PROGRAM Programm
VAR
	Alarm_Off_Time: TIME := T#3S;
	Alarm_0: Alarm;
END_VAR

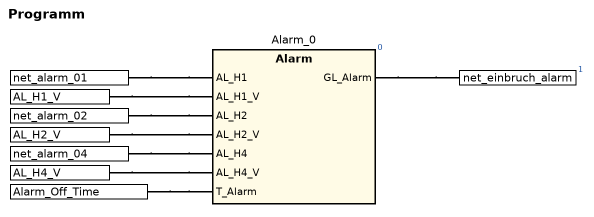
Alarm_0(
    AL_H1 := net_alarm_01,
    AL_H1_V := AL_H1_V,
    AL_H2 := net_alarm_02,
    AL_H2_V := AL_H2_V,
    AL_H4 := net_alarm_04,
    AL_H4_V := AL_H4_V,
    T_Alarm := Alarm_Off_Time); // Alarm
net_einbruch_alarm := Alarm_0.GL_Alarm;

END_PROGRAM

(* stored: Version 1.1.0.1, ProductVersion 3.1.4018.5
   POU Programm: Id {c2a23036-1c6c-4745-946e-6d5c9a463b7d}, SpecialFunc None *)
